PROGRAM MAIN
VAR
END_VAR

END_PROGRAM

(* stored: Version 1.1.0.1
   POU MAIN: Id {62c2a857-effe-4e21-a5d0-40401d1675cd} *)
